FUNCTION_BLOCK FB_Chopper_Ctrl
VAR_INPUT
	i_Interlocks		:ARRAY[1..5] OF BOOL;
	i_AutoSlowCmd		:BOOL;
	i_AutoFastCmd		:BOOL;
	i_ManSlowCmd		:BOOL;
	i_ManFastCmd		:BOOL;
	I_ManStop			:BOOL;
	i_rSpeed			:REAL;
	i_ServiceMode		:BOOL;
END_VAR
VAR_OUTPUT
	q_InterlocksOK		:BOOL;
	q_bCmdFast			:BOOL;
	q_bCmdSlow			:BOOL;
	q_rSpeed			:REAL;
END_VAR
VAR
	bCmdSlow			:BOOL;
	bCmdFast			:BOOL;
	tofSlowCMD			:TOF;
	tofFastCMD			:TOF;
	tonSlowOff			:TON;
	tonFastOff			:TON;
END_VAR
VAR // added by the converter: edge detectors and wires of the graphical bodies
    _w1 : BOOL;
END_VAR

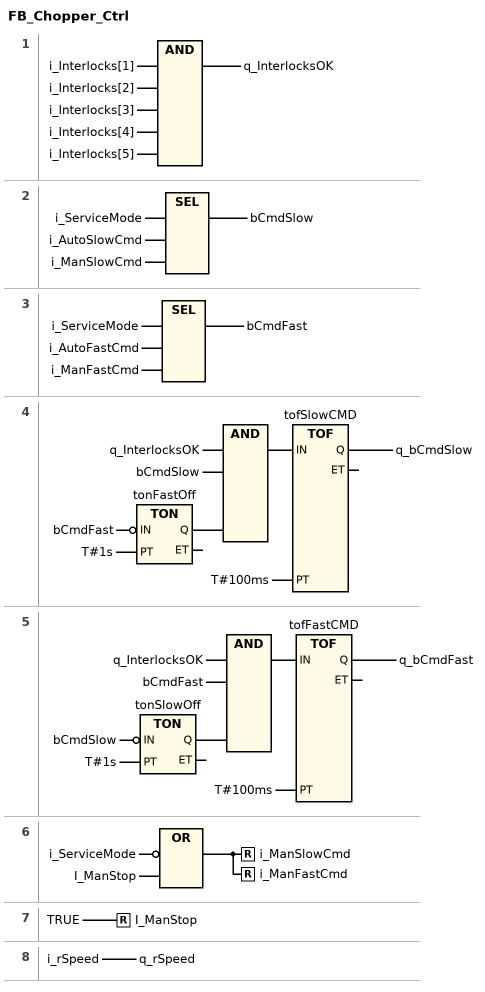
// NETWORK 1
q_InterlocksOK := i_Interlocks[1] AND i_Interlocks[2] AND i_Interlocks[3] AND i_Interlocks[4] AND i_Interlocks[5];

// NETWORK 2
bCmdSlow := SEL(i_ServiceMode, i_AutoSlowCmd, i_ManSlowCmd);

// NETWORK 3
bCmdFast := SEL(i_ServiceMode, i_AutoFastCmd, i_ManFastCmd);

// NETWORK 4
tonFastOff(IN := NOT bCmdFast, PT := T#1s); // TON
tofSlowCMD(IN := q_InterlocksOK AND bCmdSlow AND tonFastOff.Q, PT := T#100ms); // TOF
q_bCmdSlow := tofSlowCMD.Q;

// NETWORK 5
tonSlowOff(IN := NOT bCmdSlow, PT := T#1s); // TON
tofFastCMD(IN := q_InterlocksOK AND bCmdFast AND tonSlowOff.Q, PT := T#100ms); // TOF
q_bCmdFast := tofFastCMD.Q;

// NETWORK 6
_w1 := NOT i_ServiceMode OR I_ManStop;
i_ManSlowCmd R= _w1;
i_ManFastCmd R= _w1;

// NETWORK 7
I_ManStop R= TRUE;

// NETWORK 8
q_rSpeed := i_rSpeed;

END_FUNCTION_BLOCK

(* stored: Version 1.1.0.1, ProductVersion 3.1.4024.12
   POU FB_Chopper_Ctrl: Id {cf9fce54-8c1f-49ae-a090-9b002443426c}, SpecialFunc None *)
